Staubli VAL3: N10_AproBanyera.pgx

program N10_AproBanyera()
  local pointRx l_pAproBanyera
begin

  // Anar a l'aproximació del punt d'agafar líquid de la banyera
  l_pAproBanyera=pBanyera[aioGet(aiNumBanyera)]
  l_pAproBanyera.trsf.x=l_pAproBanyera.trsf.x+nXOffset
  l_pAproBanyera.trsf.y=l_pAproBanyera.trsf.y+nYOffset
  l_pAproBanyera.trsf.z=l_pAproBanyera.trsf.z+nZOffset

  if nZApro>0
    l_pAproBanyera.trsf.z=l_pAproBanyera.trsf.z+nZApro
  else
    l_pAproBanyera.trsf.z=l_pAproBanyera.trsf.z+100
  endIf

  movel(l_pAproBanyera,tToolActiva,mLent)
  waitEndMove()

  bTaskDone=true
end
